{attribute 'qualified_only'}
{attribute 'strict'}
TYPE E_Light :
(
	enum_member := 0
);
END_TYPE

(* stored: Version 1.1.0.1, ProductVersion 3.1.4024.10
   DUT E_Light: Id {f732d5a1-b02b-4190-abac-9b6cf9457683} *)
